(* IEC 61131-3 sources: repolevel_ST_code_completion/real_groud_truth最新/repoeval_Decorator_Application/full_result, 3 files *)

(* ---- ConcreteDecoratorA.st ---- *)
{attribute 'enable_dynamic_creation'}
//This class acts as a decorating class. It adds responsibilities and functionality to the component
FUNCTION_BLOCK ConcreteDecoratorA EXTENDS Decorator
VAR_INPUT
	//Reference to store the component to be decorated
	tempInputComponent : Component_Interface;
END_VAR
VAR_OUTPUT
END_VAR

VAR
	//Variable to save the state of the concrete component to be decorated
	tempComponent : Component_Interface;
	//String variable to save the Description of the component
	sDescription : STRING := 'Decorator A';
	//Real variable to save the Value of the component
	rValue : REAL;
END_VAR

METHOD getDescription : STRING
VAR_INPUT
END_VAR

//Outputs the decorated description of the component by obtaining the description of the component
// to be decorated stored in tempComponent.getDescription() and then concatenates the decoration
// description ('Decorator A' as example)
getDescription := CONCAT(THIS^.tempComponent.getDescription(), THIS^.sDescription);

METHOD getValue : REAL
VAR_INPUT
END_VAR

//Outputs the decorated value of the component by obtaining the value of the component
// to be decorated stored in tempComponent.getValue() and then adds the decoration value
getValue := THIS^.tempComponent.getValue() + THIS^.rValue;
END_FUNCTION_BLOCK

(* ---- ConcreteDecoratorB.st ---- *)
{attribute 'enable_dynamic_creation'}
//This class acts as a decorating class. It adds responsibilities and functionality to the component
FUNCTION_BLOCK ConcreteDecoratorB EXTENDS Decorator
VAR_INPUT
	//Reference to store the component to be decorated
	tempInputComponent : Component_Interface;
END_VAR
VAR_OUTPUT
END_VAR

VAR
	//Variable to save the state of the concrete component to be decorated
	tempComponent : Component_Interface;
	//String variable to save the Description of the component
	sDescription : STRING := ' Decorator B';
	//Real variable to save the Value of the component
	rValue : REAL;
END_VAR

//Method to get the decorated description of the component
METHOD getDescription : STRING
VAR_INPUT
END_VAR

//Outputs the decorated description of the component by obtaining the description of the component
// to be decorated stored in tempComponent.getDescription() and then concatenates the decoration
// description (' Decorator B' as example)
getDescription := CONCAT(THIS^.tempComponent.getDescription(), THIS^.sDescription);

//Method to get the decorated value of the component
METHOD getValue : REAL
VAR_INPUT
END_VAR

//Outputs the decorated value of the component by obtaining the value of the component
// to be decorated stored in tempComponent.getValue() and then adds the decoration value
// (e.g., adding a specific value to the original value)
getValue := THIS^.tempComponent.getValue() + THIS^.rValue;
END_FUNCTION_BLOCK

(* ---- ConcreteDecoratorC.st ---- *)
{attribute 'enable_dynamic_creation'}
//This class acts as a decorating class. It adds responsibilities and functionality to the component
FUNCTION_BLOCK ConcreteDecoratorC EXTENDS Decorator
VAR_INPUT
	//Reference to store the component to be decorated
	tempInputComponent : Component_Interface;
END_VAR
VAR_OUTPUT
END_VAR

VAR
	//Variable to save the state of the concrete component to be decorated
	tempComponent : Component_Interface;
	//String variable to save the Description of the component
	sDescription : STRING := ' Decorator C';
	//Real variable to save the Value of the component
	rValue : REAL;
END_VAR

METHOD getDescription : STRING
VAR_INPUT
	//Reference to store the component to be decorated
	tempInputComponent : Component_Interface;
END_VAR

//Outputs the decorated description of the component by obtaining the description of the component
// to be decorated stored in tempComponent.getDescription() and then concatenates the decoration
// description (' Decorator C' as example)
getDescription := CONCAT(THIS^.tempComponent.getDescription(), THIS^.sDescription);

METHOD getValue : REAL
VAR_INPUT
	//Reference to store the component to be decorated
	tempInputComponent : Component_Interface;
END_VAR

//Outputs the decorated value of the component by obtaining the value of the component
// to be decorated stored in tempComponent.getValue() and then adds the decoration value
// (e.g., adding a specific value or applying a transformation)
getValue := THIS^.tempComponent.getValue() + THIS^.rValue;
END_FUNCTION_BLOCK
